(* Schneider Machine Expert - Basic project drum-test, file version 1.9.0.0 *)
(* ProjectInformations: Name=New project *)

HARDWARE
  Cpu 0: TM221CE16R
  EthernetConfiguration: NetworkName=M221, IpAllocationMode=FixedAddress, IpAddress=0.0.0.0, SubnetMask=0.0.0.0
  SerialLineConfiguration: Baud=Baud19200, Parity=ParityEven, DataBits=DataBits8, StopBits=StopBits1, PhysicalMedium=PhysicalMediumRs485, TransmissionMode=TransmissionModeModbusRtu, SlaveId=1, Addressing=SlaveAddressing
  MastTask: UsePeriodScanMode=false, PeriodScan=100
  FastTask: Period=255
  CpuBehavior: StartingMode=StartAsPreviousState, AutoSaveRamOnEeprom=true, WatchdogPeriod=250

SYMBOLS  (address, symbol, comment, settings)

POU New POU
  (* SectionNumber=1 *)

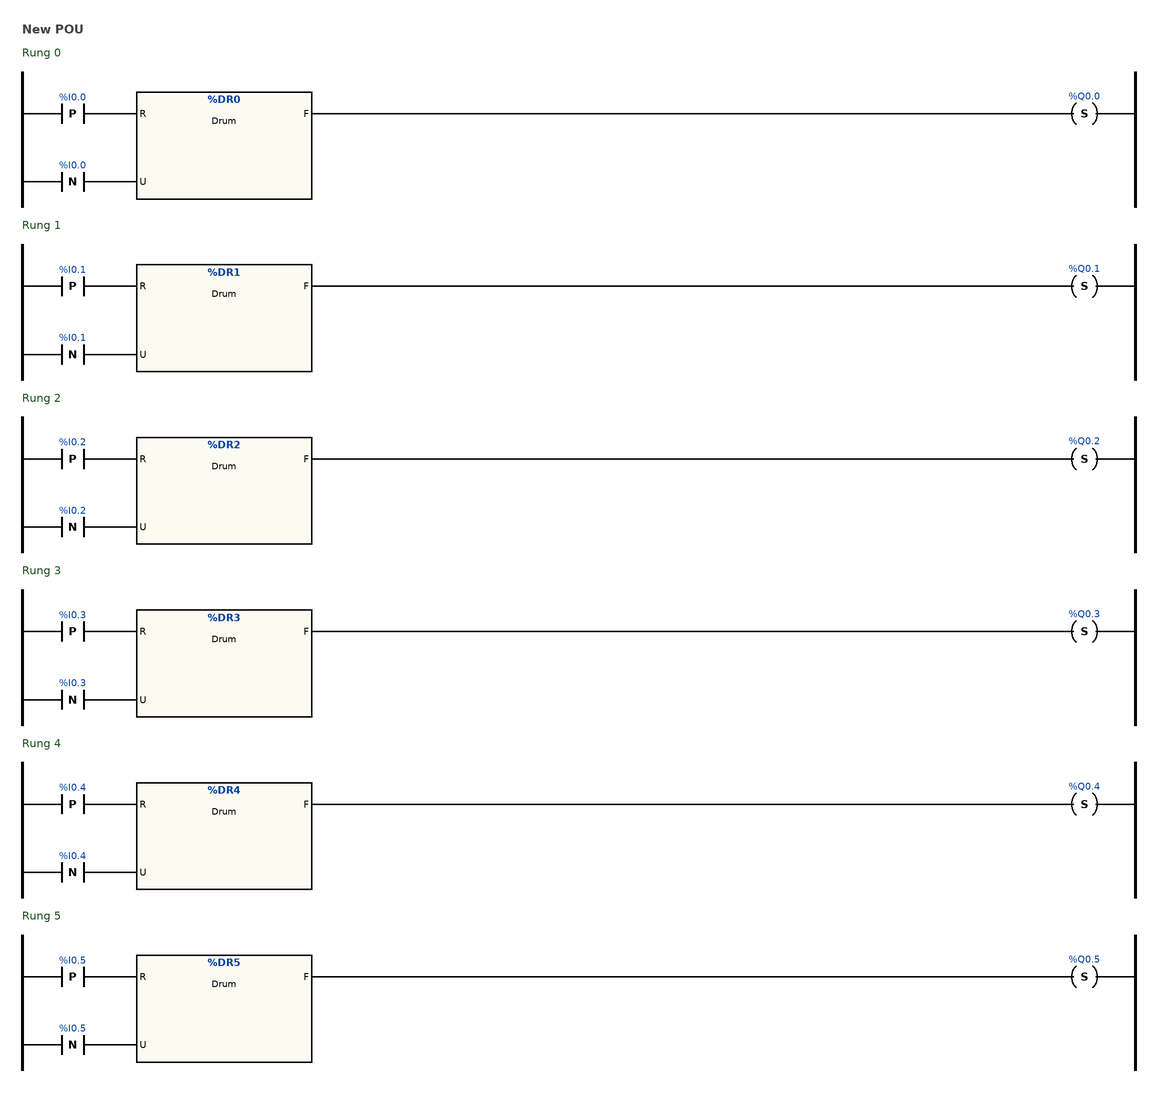

// Rung 0
  BLK %DR0
  LDR %I0.0
  R
  LDF %I0.0
  U
  OUT_BLK
  LD F
  S %Q0.0
  END_BLK
  // as ST:
  //   %DR0(R := RISING(%I0.0), U := FALLING(%I0.0));
  //   IF %DR0.F THEN %Q0.0 := TRUE; END_IF;

// Rung 1
  BLK %DR1
  LDR %I0.1
  R
  LDF %I0.1
  U
  OUT_BLK
  LD F
  S %Q0.1
  END_BLK
  // as ST:
  //   %DR1(R := RISING(%I0.1), U := FALLING(%I0.1));
  //   IF %DR1.F THEN %Q0.1 := TRUE; END_IF;

// Rung 2
  BLK %DR2
  LDR %I0.2
  R
  LDF %I0.2
  U
  OUT_BLK
  LD F
  S %Q0.2
  END_BLK
  // as ST:
  //   %DR2(R := RISING(%I0.2), U := FALLING(%I0.2));
  //   IF %DR2.F THEN %Q0.2 := TRUE; END_IF;

// Rung 3
  BLK %DR3
  LDR %I0.3
  R
  LDF %I0.3
  U
  OUT_BLK
  LD F
  S %Q0.3
  END_BLK
  // as ST:
  //   %DR3(R := RISING(%I0.3), U := FALLING(%I0.3));
  //   IF %DR3.F THEN %Q0.3 := TRUE; END_IF;

// Rung 4
  BLK %DR4
  LDR %I0.4
  R
  LDF %I0.4
  U
  OUT_BLK
  LD F
  S %Q0.4
  END_BLK
  // as ST:
  //   %DR4(R := RISING(%I0.4), U := FALLING(%I0.4));
  //   IF %DR4.F THEN %Q0.4 := TRUE; END_IF;

// Rung 5
  BLK %DR5
  LDR %I0.5
  R
  LDF %I0.5
  U
  OUT_BLK
  LD F
  S %Q0.5
  END_BLK
  // as ST:
  //   %DR5(R := RISING(%I0.5), U := FALLING(%I0.5));
  //   IF %DR5.F THEN %Q0.5 := TRUE; END_IF;

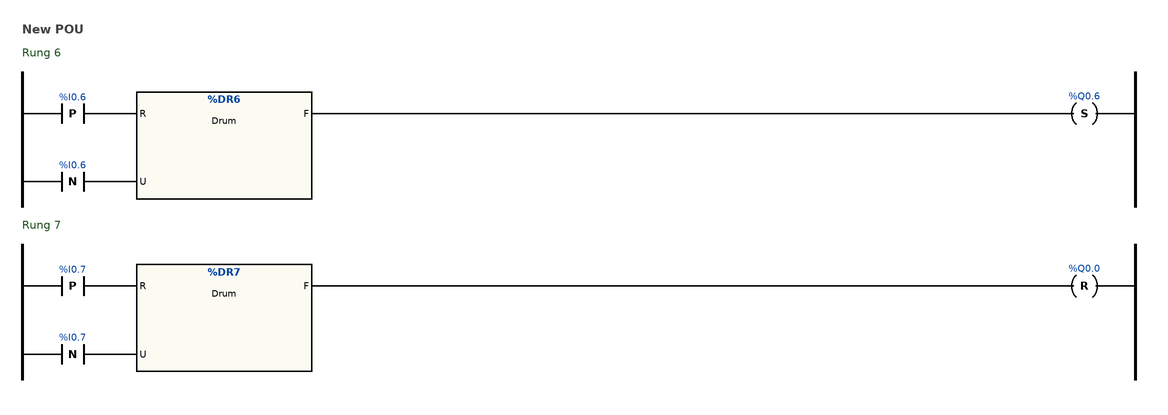

// Rung 6
  BLK %DR6
  LDR %I0.6
  R
  LDF %I0.6
  U
  OUT_BLK
  LD F
  S %Q0.6
  END_BLK
  // as ST:
  //   %DR6(R := RISING(%I0.6), U := FALLING(%I0.6));
  //   IF %DR6.F THEN %Q0.6 := TRUE; END_IF;

// Rung 7
  BLK %DR7
  LDR %I0.7
  R
  LDF %I0.7
  U
  OUT_BLK
  LD F
  R %Q0.0
  END_BLK
  // as ST:
  //   %DR7(R := RISING(%I0.7), U := FALLING(%I0.7));
  //   IF %DR7.F THEN %Q0.0 := FALSE; END_IF;
